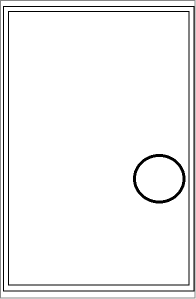
VISUALIZATION Elevator_Pause  // 196x299
    Rectangle (3,6 191x285)
    Rectangle (8,11 181x274)
    Ellipse (133,154 52x49)
    Polyline (190,297)
    Polyline (190,297)
    Polyline (119,297)
    Polyline (190,218)
    Polyline (167,217)
END_VISUALIZATION

(* stored: Version 1.1.0.1, ProductVersion 3.1.4024.12
   Visu Elevator_Pause: Id {08ada186-332b-46a5-9676-447350088be2} *)
